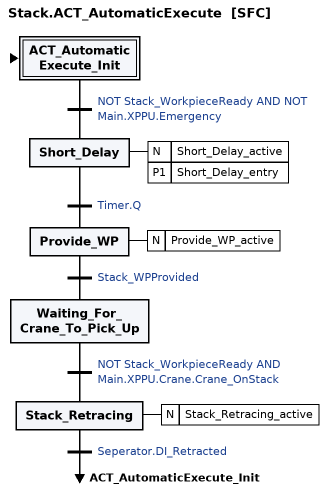
INITIAL_STEP ACT_AutomaticExecute_Init:
END_STEP
TRANSITION FROM ACT_AutomaticExecute_Init TO Short_Delay
  := NOT Stack_WorkpieceReady AND NOT Main.XPPU.Emergency;
END_TRANSITION
STEP Short_Delay:
  Short_Delay_active(N);
  Short_Delay_entry(P1);
END_STEP
TRANSITION FROM Short_Delay TO Provide_WP
  := Timer.Q;
END_TRANSITION
STEP Provide_WP:
  Provide_WP_active(N);
END_STEP
TRANSITION FROM Provide_WP TO Waiting_For_Crane_To_Pick_Up
  := Stack_WPProvided;
END_TRANSITION
STEP Waiting_For_Crane_To_Pick_Up:
END_STEP
TRANSITION FROM Waiting_For_Crane_To_Pick_Up TO Stack_Retracing
  := NOT Stack_WorkpieceReady AND Main.XPPU.Crane.Crane_OnStack;
END_TRANSITION
STEP Stack_Retracing:
  Stack_Retracing_active(N);
END_STEP
TRANSITION FROM Stack_Retracing TO ACT_AutomaticExecute_Init
  := Seperator.DI_Retracted;
END_TRANSITION
END_ACTION

ACTION ACT_Init:
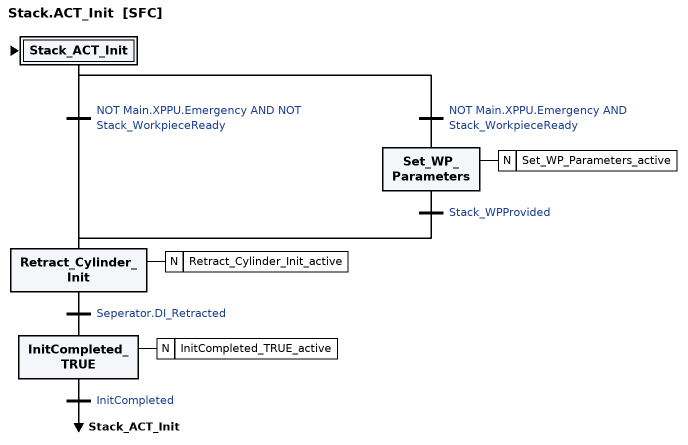
INITIAL_STEP Stack_ACT_Init:
END_STEP
TRANSITION FROM Stack_ACT_Init TO Retract_Cylinder_Init
  := NOT Main.XPPU.Emergency AND NOT Stack_WorkpieceReady;
END_TRANSITION
TRANSITION FROM Stack_ACT_Init TO Set_WP_Parameters
  := NOT Main.XPPU.Emergency AND Stack_WorkpieceReady;
END_TRANSITION
STEP Set_WP_Parameters:
  Set_WP_Parameters_active(N);
END_STEP
TRANSITION FROM Set_WP_Parameters TO Retract_Cylinder_Init
  := Stack_WPProvided;
END_TRANSITION
STEP Retract_Cylinder_Init:
  Retract_Cylinder_Init_active(N);
END_STEP
TRANSITION FROM Retract_Cylinder_Init TO InitCompleted_TRUE
  := Seperator.DI_Retracted;
END_TRANSITION
STEP InitCompleted_TRUE:
  InitCompleted_TRUE_active(N);
END_STEP
TRANSITION FROM InitCompleted_TRUE TO Stack_ACT_Init
  := InitCompleted;
END_TRANSITION
END_ACTION
END_FUNCTION_BLOCK

FUNCTION_BLOCK Stamp
VAR_INPUT
	SlidingCylinder : BistableCylinder;	
	StampingCylinder : MonostableCylinder;	
	//Software
	Stamp_SoftwareEmergency : BOOL;	
	SFCReset : BOOL;
	InitCompleted : BOOL;
	AutomaticExecuteCompleted : BOOL;
	EmergencyHandeled : BOOL;
END_VAR
VAR_OUTPUT
	//Software
	Stamp_IsStamping : BOOL;
	Stamp_WPWeight_Light : BOOL;
	Stamp_WPWeight_Medium : BOOL;
	Stamp_WPWeight_Heavy : BOOL;
	WPStamped : BOOL;
END_VAR
VAR
	//Hardware
	Stamp_SliderFilled AT %I* : BOOL;	
	Stamp_StartButton AT %I* : BOOL;
	Stamp_EmergencyStop AT %I* : BOOL;
	StampPressure AT %Q* : INT;	
	StampGreenLamp AT %Q* : BOOL;
	StampWhiteLamp AT %Q* : BOOL;
	
	//Software
	Timer : TON;
END_VAR

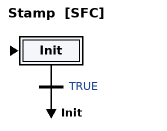
INITIAL_STEP Init:
END_STEP
TRANSITION FROM Init TO Init
  := TRUE;
END_TRANSITION

ACTION ACT_Stamp:
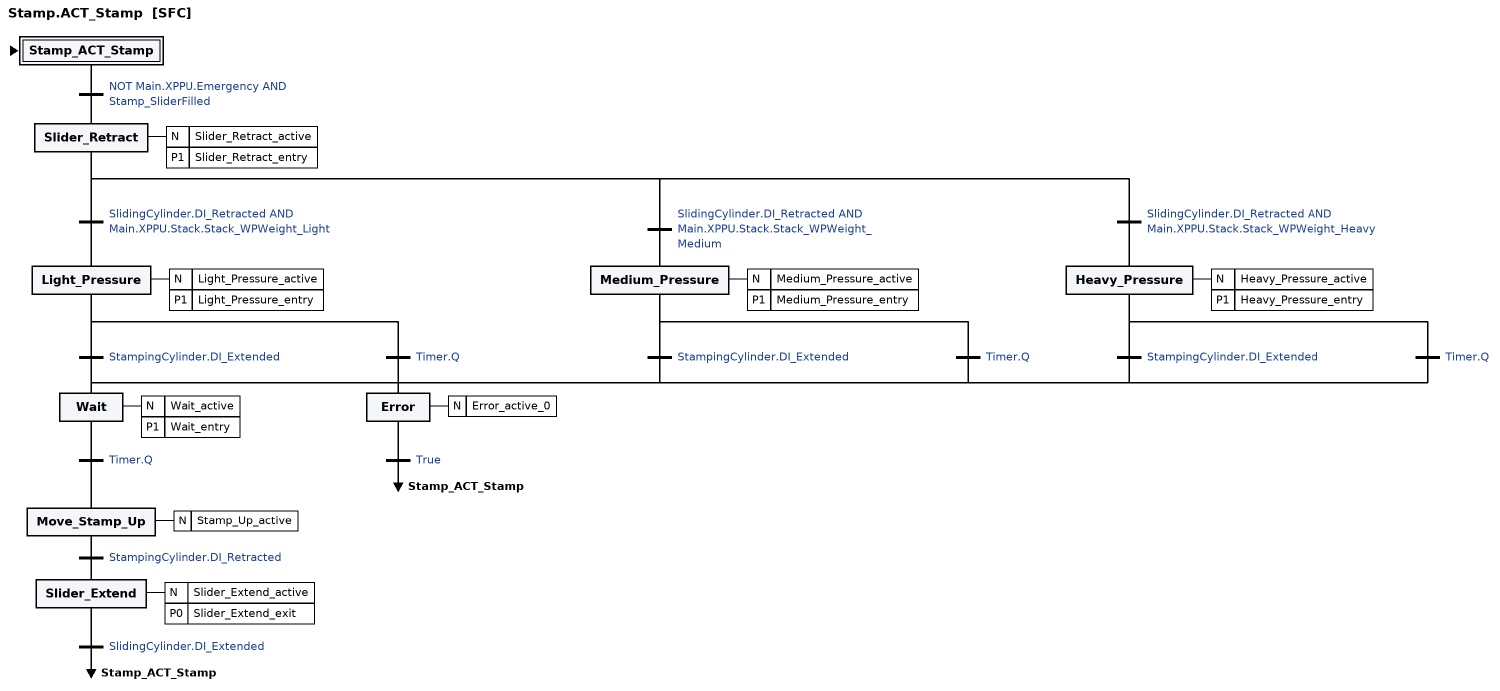
INITIAL_STEP Stamp_ACT_Stamp:
END_STEP
TRANSITION FROM Stamp_ACT_Stamp TO Slider_Retract
  := NOT Main.XPPU.Emergency AND Stamp_SliderFilled;
END_TRANSITION
STEP Slider_Retract:
  Slider_Retract_active(N);
  Slider_Retract_entry(P1);
END_STEP
TRANSITION FROM Slider_Retract TO Light_Pressure
  := SlidingCylinder.DI_Retracted AND Main.XPPU.Stack.Stack_WPWeight_Light;
END_TRANSITION
TRANSITION FROM Slider_Retract TO Medium_Pressure
  := SlidingCylinder.DI_Retracted AND Main.XPPU.Stack.Stack_WPWeight_Medium;
END_TRANSITION
TRANSITION FROM Slider_Retract TO Heavy_Pressure
  := SlidingCylinder.DI_Retracted AND Main.XPPU.Stack.Stack_WPWeight_Heavy;
END_TRANSITION
STEP Light_Pressure:
  Light_Pressure_active(N);
  Light_Pressure_entry(P1);
END_STEP
TRANSITION FROM Light_Pressure TO Wait
  := StampingCylinder.DI_Extended;
END_TRANSITION
TRANSITION FROM Light_Pressure TO Error
  := Timer.Q;
END_TRANSITION
STEP Error:
  Error_active_0(N);
END_STEP
TRANSITION FROM Error TO Stamp_ACT_Stamp
  := True;
END_TRANSITION
STEP Medium_Pressure:
  Medium_Pressure_active(N);
  Medium_Pressure_entry(P1);
END_STEP
TRANSITION FROM Medium_Pressure TO Wait
  := StampingCylinder.DI_Extended;
END_TRANSITION
TRANSITION FROM Medium_Pressure TO Error
  := Timer.Q;
END_TRANSITION
STEP Heavy_Pressure:
  Heavy_Pressure_active(N);
  Heavy_Pressure_entry(P1);
END_STEP
TRANSITION FROM Heavy_Pressure TO Wait
  := StampingCylinder.DI_Extended;
END_TRANSITION
TRANSITION FROM Heavy_Pressure TO Error
  := Timer.Q;
END_TRANSITION
STEP Wait:
  Wait_active(N);
  Wait_entry(P1);
END_STEP
TRANSITION FROM Wait TO Move_Stamp_Up
  := Timer.Q;
END_TRANSITION
STEP Move_Stamp_Up:
  Stamp_Up_active(N);
END_STEP
TRANSITION FROM Move_Stamp_Up TO Slider_Extend
  := StampingCylinder.DI_Retracted;
END_TRANSITION
STEP Slider_Extend:
  Slider_Extend_active(N);
  Slider_Extend_exit(P0);
END_STEP
TRANSITION FROM Slider_Extend TO Stamp_ACT_Stamp
  := SlidingCylinder.DI_Extended;
END_TRANSITION
END_ACTION

ACTION ACT_GreenLampOff:
                      StampGreenLamp:=FALSE;
                    
END_ACTION

ACTION ACT_GreenLampOn:
                      StampGreenLamp:=TRUE;
                    
END_ACTION

ACTION ACT_WhiteLampOff:
                      StampWhiteLamp:=FALSE;
                    
END_ACTION

ACTION ACT_WhiteLampOn:
                      StampWhiteLamp:=FALSE;
StampGreenLamp:=TRUE;
                    
END_ACTION

ACTION ACT_Init:
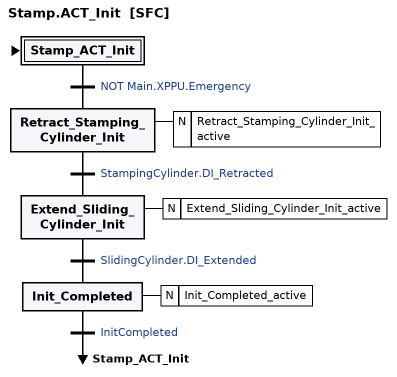
INITIAL_STEP Stamp_ACT_Init:
END_STEP
TRANSITION FROM Stamp_ACT_Init TO Retract_Stamping_Cylinder_Init
  := NOT Main.XPPU.Emergency;
END_TRANSITION
STEP Retract_Stamping_Cylinder_Init:
  Retract_Stamping_Cylinder_Init_active(N);
END_STEP
TRANSITION FROM Retract_Stamping_Cylinder_Init TO Extend_Sliding_Cylinder_Init
  := StampingCylinder.DI_Retracted;
END_TRANSITION
STEP Extend_Sliding_Cylinder_Init:
  Extend_Sliding_Cylinder_Init_active(N);
END_STEP
TRANSITION FROM Extend_Sliding_Cylinder_Init TO Init_Completed
  := SlidingCylinder.DI_Extended;
END_TRANSITION
STEP Init_Completed:
  Init_Completed_active(N);
END_STEP
TRANSITION FROM Init_Completed TO Stamp_ACT_Init
  := InitCompleted;
END_TRANSITION
END_ACTION

ACTION ACT_EmergencyStop:
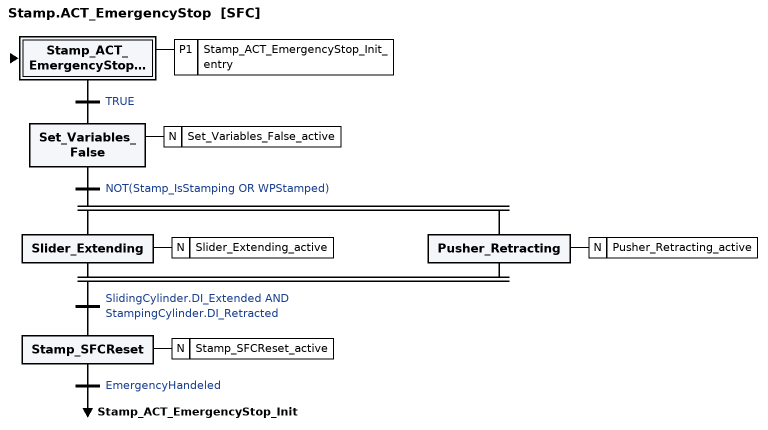
INITIAL_STEP Stamp_ACT_EmergencyStop_Init:
  Stamp_ACT_EmergencyStop_Init_entry(P1);
END_STEP
TRANSITION FROM Stamp_ACT_EmergencyStop_Init TO Set_Variables_False
  := TRUE;
END_TRANSITION
STEP Set_Variables_False:
  Set_Variables_False_active(N);
END_STEP
TRANSITION FROM Set_Variables_False TO (Slider_Extending, Pusher_Retracting)
  := NOT(Stamp_IsStamping OR WPStamped);
END_TRANSITION
STEP Slider_Extending:
  Slider_Extending_active(N);
END_STEP
TRANSITION FROM (Slider_Extending, Pusher_Retracting) TO Stamp_SFCReset
  := SlidingCylinder.DI_Extended AND StampingCylinder.DI_Retracted;
END_TRANSITION
STEP Pusher_Retracting:
  Pusher_Retracting_active(N);
END_STEP
STEP Stamp_SFCReset:
  Stamp_SFCReset_active(N);
END_STEP
TRANSITION FROM Stamp_SFCReset TO Stamp_ACT_EmergencyStop_Init
  := EmergencyHandeled;
END_TRANSITION
END_ACTION

ACTION ACT_AutomaticExecute:
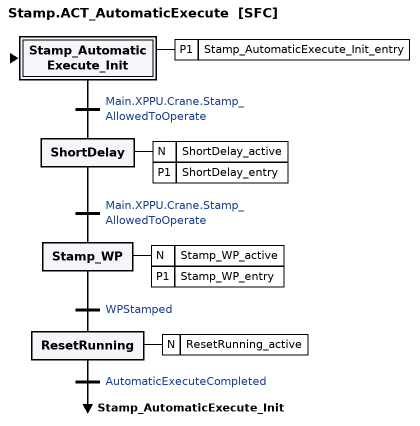
INITIAL_STEP Stamp_AutomaticExecute_Init:
  Stamp_AutomaticExecute_Init_entry(P1);
END_STEP
TRANSITION FROM Stamp_AutomaticExecute_Init TO ShortDelay
  := Main.XPPU.Crane.Stamp_AllowedToOperate;
END_TRANSITION
STEP ShortDelay:
  ShortDelay_active(N);
  ShortDelay_entry(P1);
END_STEP
TRANSITION FROM ShortDelay TO Stamp_WP
  := Main.XPPU.Crane.Stamp_AllowedToOperate;
END_TRANSITION
STEP Stamp_WP:
  Stamp_WP_active(N);
  Stamp_WP_entry(P1);
END_STEP
TRANSITION FROM Stamp_WP TO ResetRunning
  := WPStamped;
END_TRANSITION
STEP ResetRunning:
  ResetRunning_active(N);
END_STEP
TRANSITION FROM ResetRunning TO Stamp_AutomaticExecute_Init
  := AutomaticExecuteCompleted;
END_TRANSITION
END_ACTION

ACTION Error_active_0:
                      Stamp_SoftwareEmergency:=true;
                    
END_ACTION

ACTION Crane_Pick_Up_WP_active:
                      Main.XPPU.Crane.ACT_PickUpWP();
                    
END_ACTION

ACTION ResetRunning_active:
                      AutomaticExecuteCompleted:=TRUE;
                    
END_ACTION

ACTION Crane_PutWPSown_Init_active:
                      Main.XPPU.Crane.ACT_PutDownWP();
                    
END_ACTION

ACTION Stamp_Up_active:
                      StampPressure:=0;
StampingCylinder.ACT_Retract();
                    
END_ACTION

ACTION Wait_entry:
                      Timer(IN:=FALSE);
                    
END_ACTION

ACTION Wait_active:
                      Timer(IN:=True, PT:=T#1s);
                    
END_ACTION

ACTION Init_NotCompleted_active:
                      InitCompleted:=False;
                    
END_ACTION

ACTION Lower_Stamp_entry:
                      Timer(IN:=FALSE);
                    
END_ACTION

ACTION Slider_Retract_active:
                      SlidingCylinder.ACT_Retract();

Timer(IN:=TRUE, PT:=T#3s);
                    
END_ACTION

ACTION CraneToStamp_active:
                      Main.XPPU.Crane.ACT_MoveToStamp();
                    
END_ACTION

ACTION Medium_Pressure_active:
                      StampPressure:=6500;
StampingCylinder.ACT_Extend();

Timer(IN:=TRUE, PT:=T#1500MS);
                    
END_ACTION

ACTION Slider_Extend_active:
                      SlidingCylinder.ACT_Extend();

                    
END_ACTION

ACTION Stamp_SliderMoveOut_active:
                      SlidingCylinder.ACT_Extend();
                    
END_ACTION

ACTION Heavy_Pressure_active:
                      StampPressure:=7000;
StampingCylinder.ACT_Extend();

Timer(IN:=TRUE, PT:=T#1500MS);
                    
END_ACTION

ACTION Lower_Stamp_active:
                      StampingCylinder.ACT_Extend();

                    
END_ACTION

ACTION Stamp_WP_active:
                      ACT_Stamp();
                    
END_ACTION

ACTION Light_Pressure_active:
                      StampPressure:=6000;
StampingCylinder.ACT_Extend();

Timer(IN:=TRUE, PT:=T#1500MS);
                    
END_ACTION

ACTION Slider_Extending_active:
                      SlidingCylinder.ACT_Extend();
                    
END_ACTION

ACTION Stamp_WP_entry:
                      WPStamped:=FALSE;
Stamp_IsStamping:=TRUE;

                    
END_ACTION

ACTION Extend_Sliding_Cylinder_Init_active:
                      SlidingCylinder.ACT_Extend();
                    
END_ACTION

ACTION Stamp_AutomaticExecute_Init_entry:
                      AutomaticExecuteCompleted:=FALSE;
                    
END_ACTION

ACTION Stamp_ACT_EmergencyStop_Init_entry:
                      StampGreenLamp:=FALSE;
StampWhiteLamp:=FALSE;
                    
END_ACTION

ACTION MoveStampSliderOut_active:
                      SlidingCylinder.ACT_Extend();
                    
END_ACTION

ACTION Init_Completed_active:
                      InitCompleted:=TRUE;
                    
END_ACTION

ACTION Stamp_SFCReset_active:
                       EmergencyHandeled:=TRUE;	
                    
END_ACTION

ACTION Retract_Stamping_Cylinder_Init_active:
                      StampingCylinder.ACT_Retract();
                    
END_ACTION

ACTION Heavy_Pressure_entry:
                      Timer(IN:=FALSE);
                    
END_ACTION

ACTION Slider_Retract_entry:
                      Timer(IN:=FALSE);
                    
END_ACTION

ACTION Put_Wp_On_Conveyor_Init_active:
                      Main.XPPU.Crane.ACT_MoveToConveyor();
                    
END_ACTION

ACTION Medium_Pressure_entry:
                      Timer(IN:=FALSE);
                    
END_ACTION

ACTION Pusher_Retracting_active:
                      StampingCylinder.ACT_Retract();
                    
END_ACTION

ACTION SortWP_Init_active:
                      Main.XPPU.LargeSortingConveyor.ACT_SortWP();
                    
END_ACTION

ACTION Set_Variables_False_active:
                      Stamp_IsStamping:=FALSE;
WPStamped:=FALSE;
StampPressure:=0;
                    
END_ACTION

ACTION Light_Pressure_entry:
                      Timer(IN:=FALSE);
                    
END_ACTION

ACTION Slider_Extend_exit:
                      WPStamped:=TRUE;
Stamp_IsStamping:=FALSE;
                    
END_ACTION

ACTION ShortDelay_active:
                      Timer(IN:=FALSE, PT:=T#500ms);
                    
END_ACTION

ACTION ShortDelay_entry:
                      Timer(IN:=FALSE);
                    
END_ACTION
END_FUNCTION_BLOCK

FUNCTION_BLOCK XPPU
VAR_INPUT	
	//Hardware
	Stack : Stack;		
	Crane : Crane;	
	LargeSortingConveyor : LargeSortingConveyor;	
	Stamp : Stamp;
	//Software
	SFCReset : BOOL;
	StartInit : BOOL;
	Emergency : BOOL;	
END_VAR
VAR_OUTPUT
	//Software	
	InitCompleted : BOOL;
	SFCResetCompleted : BOOL;
	EmergencyHandeled : BOOL;	
END_VAR
VAR	
END_VAR

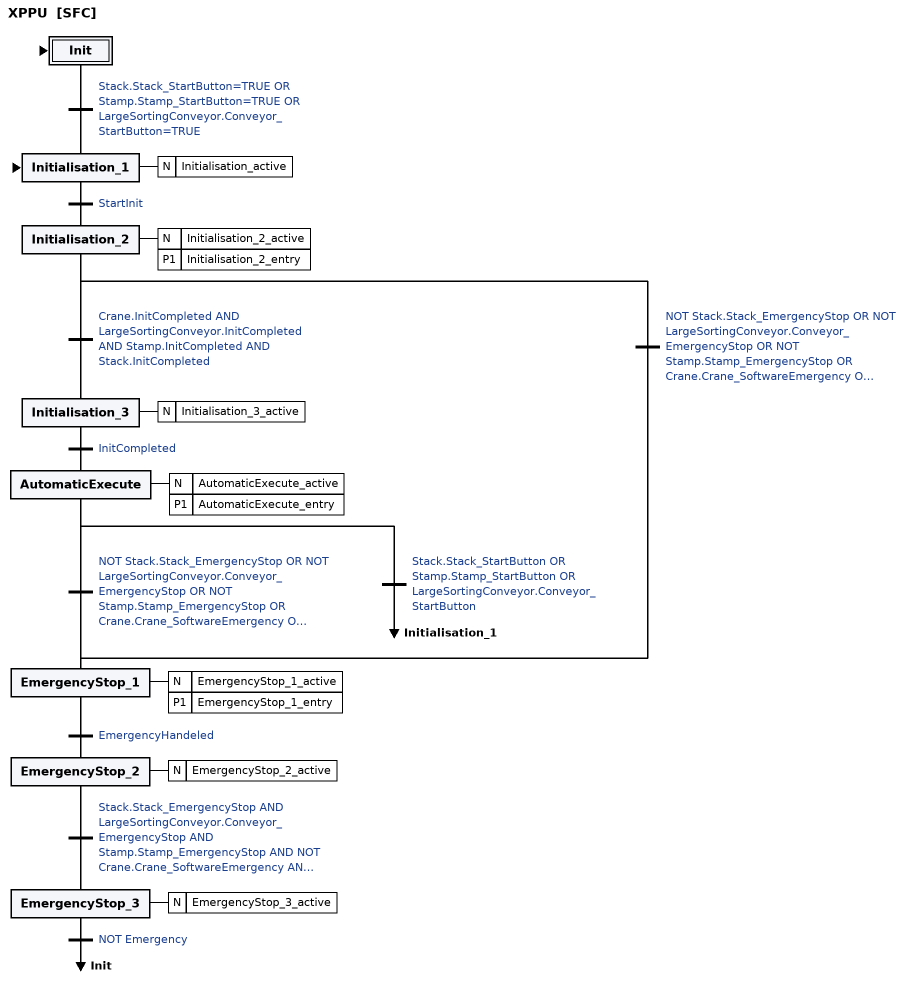
INITIAL_STEP Init:
END_STEP
TRANSITION FROM Init TO Initialisation_1
  := Stack.Stack_StartButton=TRUE OR Stamp.Stamp_StartButton=TRUE OR LargeSortingConveyor.Conveyor_StartButton=TRUE;
END_TRANSITION
STEP Initialisation_1:
  Initialisation_active(N);
END_STEP
TRANSITION FROM Initialisation_1 TO Initialisation_2
  := StartInit;
END_TRANSITION
STEP Initialisation_2:
  Initialisation_2_active(N);
  Initialisation_2_entry(P1);
END_STEP
TRANSITION FROM Initialisation_2 TO Initialisation_3
  := Crane.InitCompleted AND LargeSortingConveyor.InitCompleted AND Stamp.InitCompleted AND Stack.InitCompleted;
END_TRANSITION
TRANSITION FROM Initialisation_2 TO EmergencyStop_1
  := NOT Stack.Stack_EmergencyStop OR NOT LargeSortingConveyor.Conveyor_EmergencyStop OR NOT Stamp.Stamp_EmergencyStop OR Crane.Crane_SoftwareEmergency OR Stamp.Stamp_SoftwareEmergency;
END_TRANSITION
STEP Initialisation_3:
  Initialisation_3_active(N);
END_STEP
TRANSITION FROM Initialisation_3 TO AutomaticExecute
  := InitCompleted;
END_TRANSITION
STEP AutomaticExecute:
  AutomaticExecute_active(N);
  AutomaticExecute_entry(P1);
END_STEP
TRANSITION FROM AutomaticExecute TO EmergencyStop_1
  := NOT Stack.Stack_EmergencyStop OR NOT LargeSortingConveyor.Conveyor_EmergencyStop OR NOT Stamp.Stamp_EmergencyStop OR Crane.Crane_SoftwareEmergency OR Stamp.Stamp_SoftwareEmergency;
END_TRANSITION
TRANSITION FROM AutomaticExecute TO Initialisation_1
  := Stack.Stack_StartButton OR Stamp.Stamp_StartButton OR LargeSortingConveyor.Conveyor_StartButton;
END_TRANSITION
STEP EmergencyStop_1:
  EmergencyStop_1_active(N);
  EmergencyStop_1_entry(P1);
END_STEP
TRANSITION FROM EmergencyStop_1 TO EmergencyStop_2
  := EmergencyHandeled;
END_TRANSITION
STEP EmergencyStop_2:
  EmergencyStop_2_active(N);
END_STEP
TRANSITION FROM EmergencyStop_2 TO EmergencyStop_3
  := Stack.Stack_EmergencyStop AND LargeSortingConveyor.Conveyor_EmergencyStop AND Stamp.Stamp_EmergencyStop AND NOT Crane.Crane_SoftwareEmergency AND NOT Stamp.Stamp_SoftwareEmergency;
END_TRANSITION
STEP EmergencyStop_3:
  EmergencyStop_3_active(N);
END_STEP
TRANSITION FROM EmergencyStop_3 TO Init
  := NOT Emergency;
END_TRANSITION

ACTION ACT_EmergencyStop:
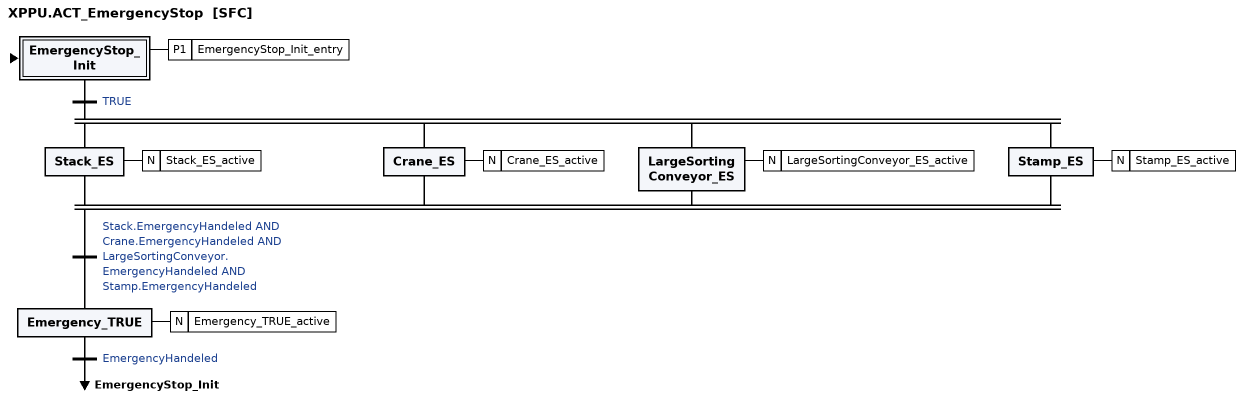
INITIAL_STEP EmergencyStop_Init:
  EmergencyStop_Init_entry(P1);
END_STEP
TRANSITION FROM EmergencyStop_Init TO (Stack_ES, Crane_ES, LargeSortingConveyor_ES, Stamp_ES)
  := TRUE;
END_TRANSITION
STEP Stack_ES:
  Stack_ES_active(N);
END_STEP
TRANSITION FROM (Stack_ES, Crane_ES, LargeSortingConveyor_ES, Stamp_ES) TO Emergency_TRUE
  := Stack.EmergencyHandeled AND Crane.EmergencyHandeled AND LargeSortingConveyor.EmergencyHandeled AND Stamp.EmergencyHandeled;
END_TRANSITION
STEP Crane_ES:
  Crane_ES_active(N);
END_STEP
STEP LargeSortingConveyor_ES:
  LargeSortingConveyor_ES_active(N);
END_STEP
STEP Stamp_ES:
  Stamp_ES_active(N);
END_STEP
STEP Emergency_TRUE:
  Emergency_TRUE_active(N);
END_STEP
TRANSITION FROM Emergency_TRUE TO EmergencyStop_Init
  := EmergencyHandeled;
END_TRANSITION
END_ACTION

ACTION ACT_AutomaticExecute:
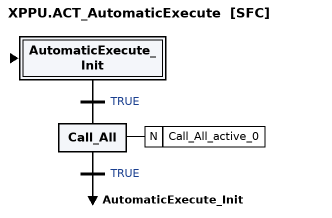
INITIAL_STEP AutomaticExecute_Init:
END_STEP
TRANSITION FROM AutomaticExecute_Init TO Call_All
  := TRUE;
END_TRANSITION
STEP Call_All:
  Call_All_active_0(N);
END_STEP
TRANSITION FROM Call_All TO AutomaticExecute_Init
  := TRUE;
END_TRANSITION
END_ACTION

ACTION ACT_Init:
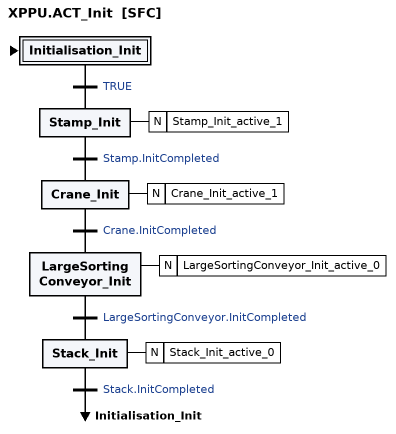
INITIAL_STEP Initialisation_Init:
END_STEP
TRANSITION FROM Initialisation_Init TO Stamp_Init
  := TRUE;
END_TRANSITION
STEP Stamp_Init:
  Stamp_Init_active_1(N);
END_STEP
TRANSITION FROM Stamp_Init TO Crane_Init
  := Stamp.InitCompleted;
END_TRANSITION
STEP Crane_Init:
  Crane_Init_active_1(N);
END_STEP
TRANSITION FROM Crane_Init TO LargeSortingConveyor_Init
  := Crane.InitCompleted;
END_TRANSITION
STEP LargeSortingConveyor_Init:
  LargeSortingConveyor_Init_active_0(N);
END_STEP
TRANSITION FROM LargeSortingConveyor_Init TO Stack_Init
  := LargeSortingConveyor.InitCompleted;
END_TRANSITION
STEP Stack_Init:
  Stack_Init_active_0(N);
END_STEP
TRANSITION FROM Stack_Init TO Initialisation_Init
  := Stack.InitCompleted;
END_TRANSITION
END_ACTION

ACTION Crane_Init_active_1:
                      Crane.ACT_Init();
                    
END_ACTION

ACTION EmergencyStop_3_active:
                      Emergency:=FALSE;
                    
END_ACTION

ACTION LargeSortingConveyor_Init_active:
                      LargeSortingConveyor.ACT_Init();
                    
END_ACTION

ACTION Crane_ES_active:
                      Crane.ACT_EmergencyStop();
                    
END_ACTION

ACTION Stack_Init_active:
                      Stack.ACT_Init();
                    
END_ACTION

ACTION LargeSortingConveyor_Init_active_0:
                      LargeSortingConveyor.ACT_Init();
                    
END_ACTION

ACTION Stamp_Init_active:
                      Stamp.ACT_Init();
                    
END_ACTION

ACTION Call_All_active_0:
                      Stack.ACT_AutomaticExecute();
Crane.ACT_AutomaticExecute();
Stamp.ACT_AutomaticExecute();
LargeSortingConveyor.ACT_AutomaticExecute();
                    
END_ACTION

ACTION Stack_Init_active_0:
                      Stack.ACT_Init();
                    
END_ACTION

ACTION Stack_ES_active:
                      Stack.ACT_EmergencyStop();
                    
END_ACTION

ACTION Stamp_Init_active_1:
                      Stamp.ACT_Init();
                    
END_ACTION

ACTION Initialisation_3_active:
                      StartInit:=FALSE;
InitCompleted:=TRUE;
                    
END_ACTION

ACTION Stamp_Init_active_0:
                      Stamp.ACT_Init();
                    
END_ACTION

ACTION EmergencyStop_2_active:
                      (*Stack Reset*)
Stack.ACT_AutomaticExecute(SFCReset:=TRUE);
Stack.ACT_Init(SFCReset:=TRUE);
Stack.ACT_ProvideWP(SFCReset:=TRUE);
//Stack.Seperator.ACT_Extend(SFCREset:=TRUE);
//Stack.Seperator.ACT_Retract(SFCREset:=TRUE);		
(*Crane Reset*)
Crane.ACT_AutomaticExecute(SFCReset:=TRUE);
Crane.ACT_Init(SFCReset:=TRUE);
Crane.ACT_MoveToConveyor(SFCReset:=TRUE);
Crane.ACT_MoveToStack(SFCReset:=TRUE);
Crane.ACT_MoveToStamp(SFCReset:=TRUE);
Crane.ACT_PickUpWP(SFCReset:=TRUE);
Crane.ACT_PutDownWP(SFCReset:=TRUE);
//Crane.LiftingCylinder.ACT_Extend(SFCREset:=TRUE);	
//Crane.LiftingCylinder.ACT_Retract(SFCREset:=TRUE);
//Crane.Gripper.ACT_Intake(SFCREset:=TRUE);
//Crane.Gripper.ACT_Release(SFCREset:=TRUE);	
(*LargeSortingConveyor Reset*)
LargeSortingConveyor.ACT_ChangeTarget(SFCReset:=TRUE);
LargeSortingConveyor.ACT_CheckWPType(SFCReset:=TRUE);
LargeSortingConveyor.ACT_Init(SFCReset:=TRUE);
LargeSortingConveyor.ACT_SortWP(SFCReset:=TRUE);
//LargeSortingConveyor.Motor.ACT_Stop(SFCREset:=TRUE);
//LargeSortingConveyor.Motor.ACT_TurnBackwards(SFCREset:=TRUE);
//LargeSortingConveyor.Motor.ACT_TurnForwards(SFCREset:=TRUE);
//LargeSortingConveyor.SwitchPicAlpha.ACT_Extend(SFCREset:=TRUE);
//LargeSortingConveyor.SwitchPicAlpha.ACT_Retract(SFCREset:=TRUE);
//LargeSortingConveyor.Seperator1.ACT_Retract(SFCREset:=TRUE);
//LargeSortingConveyor.Seperator2.ACT_Extend(SFCREset:=TRUE);
//LargeSortingConveyor.Seperator2.ACT_Retract(SFCREset:=TRUE);
(*Stamp Reset*)
Stamp.ACT_Init(SFCReset:=TRUE);
Stamp.ACT_Stamp(SFCReset:=TRUE);
//Stamp.SlidingCylinder.ACT_Extend(SFCREset:=TRUE);
//Stamp.SlidingCylinder.ACT_Retract(SFCREset:=TRUE);
//Stamp.StampingCylinder.ACT_Extend(SFCREset:=TRUE);
//Stamp.StampingCylinder.ACT_Retract(SFCREset:=TRUE);

IF(Stack.Stack_StartButton=TRUE OR Stamp.Stamp_StartButton=TRUE OR LargeSortingConveyor.Conveyor_StartButton=TRUE)THEN
	Stamp.Stamp_SoftwareEmergency:=FALSE;
	Crane.Crane_SoftwareEmergency:=FALSE;
END_IF	

SFCResetCompleted:=TRUE;	
                    
END_ACTION

ACTION EmergencyStop_Init_entry:
                      EmergencyHandeled:=FALSE;
                    
END_ACTION

ACTION EmergencyStop_1_active:
                      ACT_EmergencyStop(); 	
	
InitCompleted:=FALSE;
Stack.InitCompleted:=FALSE;
Crane.InitCompleted:=FALSE;
Stamp.InitCompleted:=FALSE;
LargeSortingConveyor.InitCompleted:=FALSE;
                    
END_ACTION

ACTION AutomaticExecute_active:
                      ACT_AutomaticExecute();
                    
END_ACTION

ACTION Initialisation_2_entry:
                      LargeSortingConveyor.ACT_WhiteLampOn();
Stack.ACT_WhiteLampOn();	
Stamp.ACT_WhiteLampOn();
LargeSortingConveyor.ACT_GreenLampOff();
Stack.ACT_GreenLampOff();	
Stamp.ACT_GreenLampOff();
                    
END_ACTION

ACTION LargeSortingConveyor_Init2_active:
                      LargeSortingConveyor.ACT_Init();
                    
END_ACTION

ACTION Emergency_TRUE_active:
                      EmergencyHandeled:=TRUE;
                    
END_ACTION

ACTION Initialisation_2_active:
                      ACT_Init();
                    
END_ACTION

ACTION AutomaticExecute_entry:
                      LargeSortingConveyor.ACT_WhiteLampOff();
Stack.ACT_WhiteLampOff();	
Stamp.ACT_WhiteLampOff();
LargeSortingConveyor.ACT_GreenLampOn();
Stack.ACT_GreenLampOn();	
Stamp.ACT_GreenLampOn();
                    
END_ACTION

ACTION Stamp_ES_active:
                      Stamp.ACT_EmergencyStop();
                    
END_ACTION

ACTION Crane_Init_active:
                      Crane.ACT_Init();
                    
END_ACTION

ACTION Initialisation_active:
                      Crane.Crane_SoftwareEmergency:=FALSE;
Stamp.Stamp_SoftwareEmergency:=FALSE;

Crane.InitCompleted:=FALSE;
LargeSortingConveyor.InitCompleted:=FALSE;
Stamp.InitCompleted:=FALSE;
Stack.InitCompleted:=FALSE;
InitCompleted:=FALSE;

(*Stack Reset*)
Stack.ACT_AutomaticExecute(SFCReset:=FALSE);
Stack.ACT_Init(SFCReset:=FALSE);
Stack.ACT_ProvideWP(SFCReset:=FALSE);
//Stack.Seperator.ACT_Extend(SFCREset:=FALSE);
//Stack.Seperator.ACT_Retract(SFCREset:=FALSE);		
(*Crane Reset*)
Crane.ACT_AutomaticExecute(SFCReset:=FALSE);
Crane.ACT_Init(SFCReset:=FALSE);
Crane.ACT_MoveToConveyor(SFCReset:=FALSE);
Crane.ACT_MoveToStack(SFCReset:=FALSE);
Crane.ACT_MoveToStamp(SFCReset:=FALSE);
Crane.ACT_PickUpWP(SFCReset:=FALSE);
Crane.ACT_PutDownWP(SFCReset:=FALSE);
//Crane.LiftingCylinder.ACT_Extend(SFCREset:=FALSE);	
//Crane.LiftingCylinder.ACT_Retract(SFCREset:=FALSE);
//Crane.Gripper.ACT_Intake(SFCREset:=FALSE);
//Crane.Gripper.ACT_Release(SFCREset:=FALSE);	
(*LargeSortingConveyor Reset*)
LargeSortingConveyor.ACT_ChangeTarget(SFCReset:=FALSE);
LargeSortingConveyor.ACT_CheckWPType(SFCReset:=FALSE);
LargeSortingConveyor.ACT_Init(SFCReset:=FALSE);
LargeSortingConveyor.ACT_SortWP(SFCReset:=FALSE);
//LargeSortingConveyor.Motor.ACT_Stop(SFCREset:=FALSE);
//LargeSortingConveyor.Motor.ACT_TurnBackwards(SFCREset:=FALSE);
//LargeSortingConveyor.Motor.ACT_TurnForwards(SFCREset:=FALSE);
//LargeSortingConveyor.SwitchPicAlpha.ACT_Extend(SFCREset:=FALSE);
//LargeSortingConveyor.SwitchPicAlpha.ACT_Retract(SFCREset:=FALSE);
//LargeSortingConveyor.Seperator1.ACT_Retract(SFCREset:=FALSE);
//LargeSortingConveyor.Seperator2.ACT_Extend(SFCREset:=FALSE);
//LargeSortingConveyor.Seperator2.ACT_Retract(SFCREset:=FALSE);
(*Stamp Reset*)
Stamp.ACT_Init(SFCReset:=FALSE);
Stamp.ACT_Stamp(SFCReset:=FALSE);
//Stamp.SlidingCylinder.ACT_Extend(SFCREset:=FALSE);
//Stamp.SlidingCylinder.ACT_Retract(SFCREset:=FALSE);
//Stamp.StampingCylinder.ACT_Extend(SFCREset:=FALSE);
//Stamp.StampingCylinder.ACT_Retract(SFCREset:=FALSE);

SFCResetCompleted:=FALSE;	

StartInit:=TRUE;	
                    
END_ACTION

ACTION LargeSortingConveyor_ES_active:
                      LargeSortingConveyor.ACT_EmergencyStop();
                    
END_ACTION

ACTION EmergencyStop_1_entry:
                      Emergency:=TRUE;

LargeSortingConveyor.ACT_WhiteLampOff();
Stack.ACT_WhiteLampOff();	
Stamp.ACT_WhiteLampOff();
LargeSortingConveyor.ACT_GreenLampOff();
Stack.ACT_GreenLampOff();	
Stamp.ACT_GreenLampOff();
                    
END_ACTION

ACTION Crane_Init_active_0:
                      Crane.ACT_Init();
                    
END_ACTION
END_FUNCTION_BLOCK

CONFIGURATION Application
  RESOURCE project ON PLC
    TASK PlcTask(INTERVAL := T#0ms, PRIORITY := 22);
    PROGRAM MAIN WITH PlcTask : MAIN;
  END_RESOURCE
END_CONFIGURATION
